// TIA Portal V16 export
// export: Created 2025-08-30T12:59:11.5374767Z, ExportSetting WithDefaults, DisplayName Totally Integrated Automation Portal, DisplayVersion V16, DisplayName TIA Portal Version Control Interface, DisplayVersion V16, DisplayName TIA Portal Openness, DisplayVersion V16, DisplayName STEP 7 Professional, DisplayVersion V16, DisplayName STEP 7 Safety, DisplayVersion V16, DisplayName WinCC Advanced, DisplayVersion V16
FUNCTION_BLOCK "FB_EncoderFeedback_Lineair"   // FB21, FBD
TITLE = Encoder Feedback Function Block Lineair Axis
VERSION : 0.1
// stored: AutoNumber true, IsIECCheckEnabled false, UDAEnableTagReadback false
   VAR_INPUT
      CounterTag { ExternalVisible := 'False'; ExternalWritable := 'False'} : DInt;   // Connect to the CounterTag IW102
      Position_Offset { ExternalVisible := 'False'; ExternalWritable := 'False'} : Real;   // Fill in the tolerance, when the axis approves the position. Above or below the desired position
      Pulsfactor { ExternalVisible := 'False'; ExternalWritable := 'False'} : Real;   // Number of pulses after an defined distance of the axis.
      Position_Correction { ExternalVisible := 'False'; ExternalWritable := 'False'} : Real;   // Small Position Correction for the Axis
      ReferenceRun_Command { ExternalVisible := 'False'; ExternalWritable := 'False'} : Bool;   // Command of starting the referencerun
      ReferenceSwitch { ExternalVisible := 'False'; ExternalWritable := 'False'} : Bool;   // ReferenceSwitch Mounted on Axis
      ReferencePosition { ExternalVisible := 'False'; ExternalWritable := 'False'} : Int;   // Position where the index puls of the reference switch enters.
      WrappingPosition : Real;   // Max Position of the axis. From there the position
   END_VAR
   VAR_OUTPUT
      Scaled_Position { ExternalVisible := 'False'; ExternalWritable := 'False'} : Real;   // Scaled Position scaled with Pulsfactor
      Actual_Enc_Pos { ExternalVisible := 'False'; ExternalWritable := 'False'} : Real;   // Actual Encoder Position
      AxisDB_Connection { ExternalVisible := 'False'; ExternalWritable := 'False'} : Real;   // Connection with Axis DB connection
   END_VAR
   VAR_TEMP
      Corrected_Axis_Pos : Real;
      Unscaled_Position : DInt;   // Unscaled Position of the Encoder
      Unsc2 : DInt;   // Unsc 2 position
      Act_Enc_Pos_Int : DInt;
      Scaled_Position_Real : Real;
      PosDint : DInt;
      Unscaled_Position_Real : Real;
      InternalCounter : DInt;
      CalDifCounter : DInt;
      Pos_Storage : DInt;
      Pos_Diffrence : DInt;
      Add_Pos : DInt;
      Sub_Pos : DInt;
      LessThanZero : Bool;
      LTZ_out : DInt;
      WrappedPosTemp : Real;
      DivWrapping : Real;
      TruncWrapping : DInt;
      TruncWrappingReal : Real;
      ScaledBackWrapping : Real;
      AxisPosTooHigh : Bool;
      WeDontUseThisAnymore : Bool;
      SRMOve : Bool;
      noreset : Bool;
      nououtput : Bool;
      OverflowProtectPulses : DInt;
      SegmentCounter : DInt;
   END_VAR
BEGIN

REGION Network 1: Overflow Buffer FB
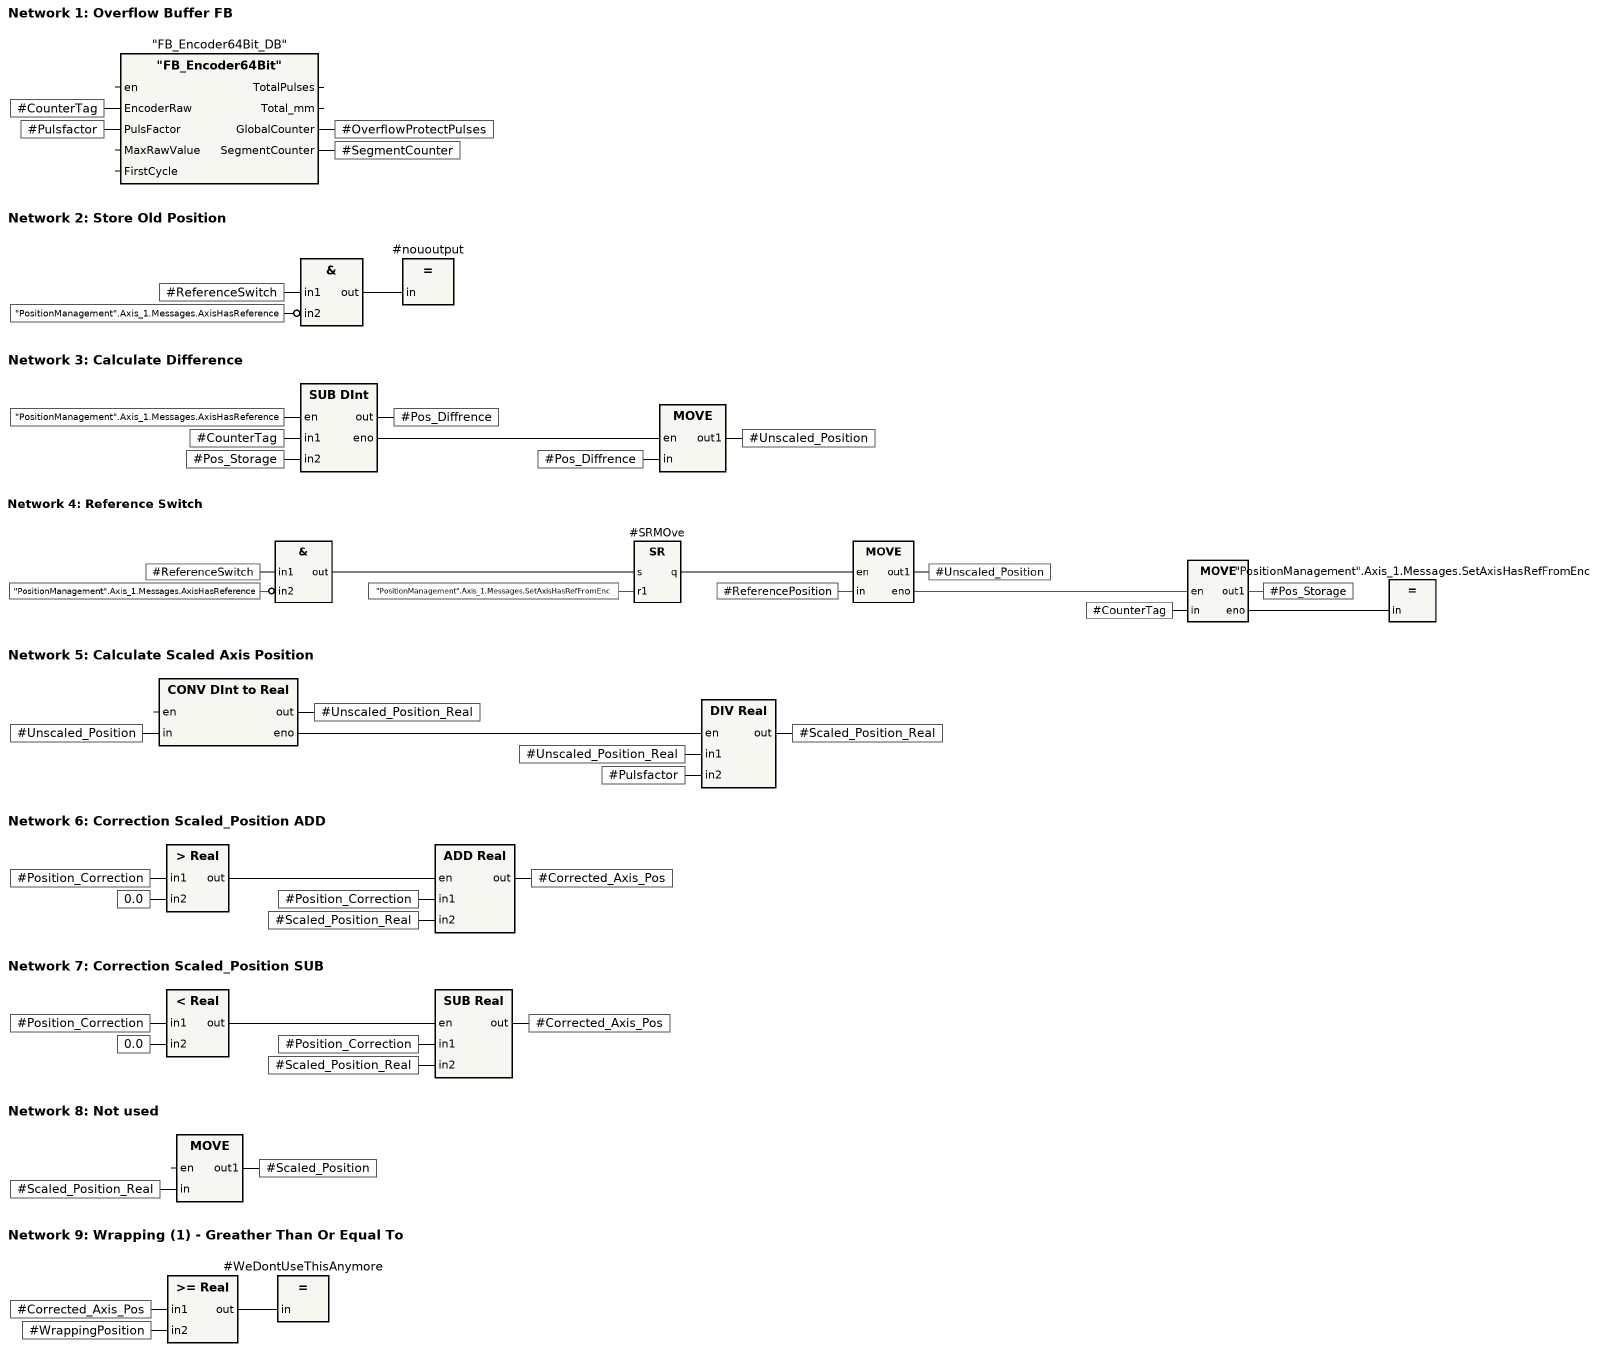
   "FB_Encoder64Bit_DB"(EncoderRaw := #CounterTag,   // "FB_Encoder64Bit"
                        PulsFactor := #Pulsfactor,
                        GlobalCounter => #OverflowProtectPulses,
                        SegmentCounter => #SegmentCounter);
END_REGION

REGION Network 2: Store Old Position
   #nououtput := #ReferenceSwitch AND NOT "PositionManagement".Axis_1.Messages.AxisHasReference;
END_REGION

REGION Network 3: Calculate Difference
   // ENO of a box is taken as its EN; it also drops when the box reports an error
   IF "PositionManagement".Axis_1.Messages.AxisHasReference THEN
       #Pos_Diffrence := #CounterTag - #Pos_Storage;
       #Unscaled_Position := #Pos_Diffrence;
   END_IF;
END_REGION

REGION Network 4: Reference Switch
   // ENO of a box is taken as its EN; it also drops when the box reports an error
   IF #ReferenceSwitch AND NOT "PositionManagement".Axis_1.Messages.AxisHasReference THEN
       #SRMOve := TRUE;   // SR flip-flop
   END_IF;
   IF "PositionManagement".Axis_1.Messages.SetAxisHasRefFromEnc THEN #SRMOve := FALSE; END_IF;
   IF #SRMOve THEN
       #Unscaled_Position := #ReferencePosition;
       #Pos_Storage := #CounterTag;
   END_IF;
   "PositionManagement".Axis_1.Messages.SetAxisHasRefFromEnc := #SRMOve;
END_REGION

REGION Network 5: Calculate Scaled Axis Position
   // ENO of a box is taken as its EN; it also drops when the box reports an error
   #Unscaled_Position_Real := DINT_TO_REAL(#Unscaled_Position);
   #Scaled_Position_Real := #Unscaled_Position_Real / #Pulsfactor;
END_REGION

REGION Network 6: Correction Scaled_Position ADD
   IF #Position_Correction > 0.0 THEN
       #Corrected_Axis_Pos := #Position_Correction + #Scaled_Position_Real;
   END_IF;
END_REGION

REGION Network 7: Correction Scaled_Position SUB
   IF #Position_Correction < 0.0 THEN
       #Corrected_Axis_Pos := #Position_Correction - #Scaled_Position_Real;
   END_IF;
END_REGION

REGION Network 8: Not used
   #Scaled_Position := #Scaled_Position_Real;
END_REGION

REGION Network 9: Wrapping (1) - Greather Than Or Equal To
   #WeDontUseThisAnymore := #Corrected_Axis_Pos >= #WrappingPosition;
END_REGION

REGION Network 10: Wrapping (2) - MOVE Axis Pos Too High
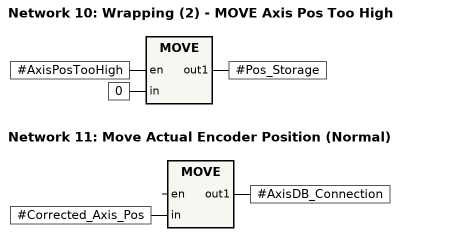
   IF #AxisPosTooHigh THEN #Pos_Storage := 0; END_IF;
END_REGION

REGION Network 11: Move Actual Encoder Position (Normal)
   #AxisDB_Connection := #Corrected_Axis_Pos;
END_REGION
END_FUNCTION_BLOCK
